FUNCTION_BLOCK DataPanel_xDB_16_ADI_SAE_J1939 (* Service Interface Function Block Type *)
  (* Standard: SAE J1939; Function: All Inputs; Type: DP-34044-2-000; Description: Copyright (c) 2018, 2023 Jose Cabral, HR Agrartechnik GmbH This program and the accompanying materials are made available under the terms of the Eclipse Public License 2.0 which is available at https://www.eclipse.org/legal/epl-2.0/ SPDX-License-Identifier: EPL-2.0 this maps to IX *)
  (* Version 1.0, 2018-12-05, Jose Cabral *)
  (* Version 1.1, 2022-08-04, Franz Höpfinger, HR Agrartechnik GmbH *)
  (* Version 1.2, 2023-01-05, Franz Höpfinger, HR Agrartechnik GmbH *)
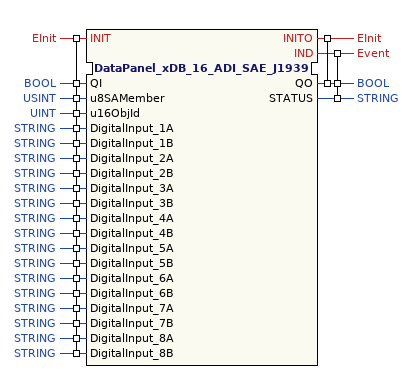
  EVENT_INPUT
    INIT : EInit WITH QI, u8SAMember, u16ObjId, DigitalInput_1A, DigitalInput_1B, DigitalInput_2A, DigitalInput_2B, DigitalInput_3A, DigitalInput_3B, DigitalInput_4A, DigitalInput_4B, DigitalInput_5A, DigitalInput_5B, DigitalInput_6A, DigitalInput_6B, DigitalInput_7A, DigitalInput_7B, DigitalInput_8A, DigitalInput_8B; (* Service Initialization *)
  END_EVENT
  EVENT_OUTPUT
    INITO : EInit WITH QO; (* Initialization Confirm *)
    IND WITH QO, STATUS; (* Indication from Resource *)
  END_EVENT
  VAR_INPUT
    QI : BOOL; (* Event Input Qualifier *)
    u8SAMember : USINT := MI::MI_00; (* Node SA 224..239 *)
    u16ObjId : UINT := isobus::ID_NULL; (* Dummy ! set to ID_NULL if in Doubt. ID_OFF deactivates FB. *)
    DigitalInput_1A : STRING;
    DigitalInput_1B : STRING;
    DigitalInput_2A : STRING;
    DigitalInput_2B : STRING;
    DigitalInput_3A : STRING;
    DigitalInput_3B : STRING;
    DigitalInput_4A : STRING;
    DigitalInput_4B : STRING;
    DigitalInput_5A : STRING;
    DigitalInput_5B : STRING;
    DigitalInput_6A : STRING;
    DigitalInput_6B : STRING;
    DigitalInput_7A : STRING;
    DigitalInput_7B : STRING;
    DigitalInput_8A : STRING;
    DigitalInput_8B : STRING;
  END_VAR
  VAR_OUTPUT
    QO : BOOL; (* Event Output Qualifier *)
    STATUS : STRING; (* Service Status *)
  END_VAR
END_FUNCTION_BLOCK
